// Mitsubishi GX Works2 project: LD_windingmachine   PLC: FX1N/FX1NC

PROGRAM MAIN
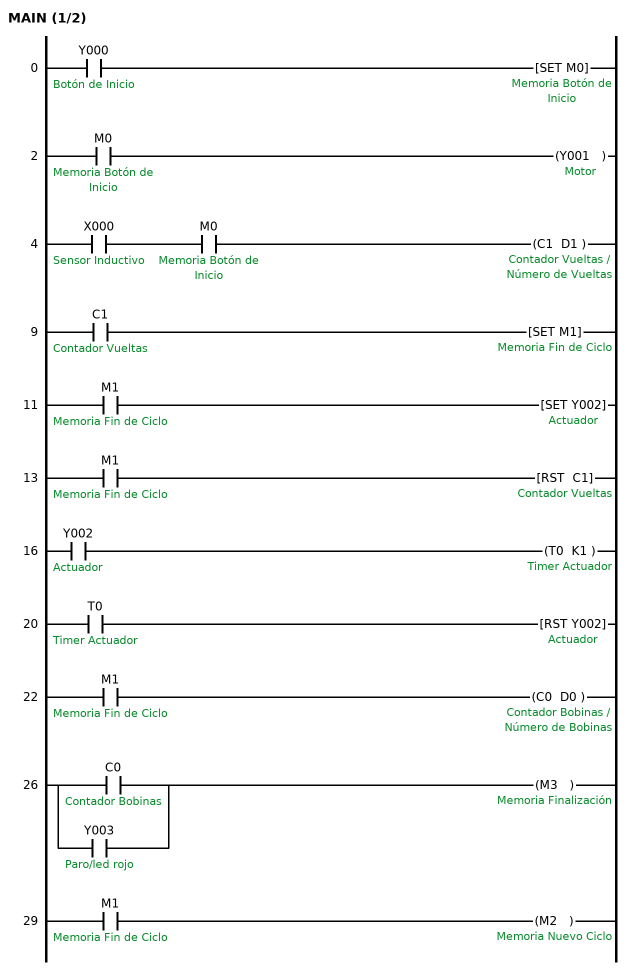
0     LD      Y000  ; Botón de Inicio
      SET     M0  ; Memoria Botón de Inicio
2     LD      M0  ; Memoria Botón de Inicio
      OUT     Y001  ; Motor
4     LD      X000  ; Sensor Inductivo
      AND     M0  ; Memoria Botón de Inicio
      OUT     C1 D1  ; Contador Vueltas / Número de Vueltas
9     LD      C1  ; Contador Vueltas
      SET     M1  ; Memoria Fin de Ciclo
11    LD      M1  ; Memoria Fin de Ciclo
      SET     Y002  ; Actuador
13    LD      M1  ; Memoria Fin de Ciclo
      RST     C1  ; Contador Vueltas
16    LD      Y002  ; Actuador
      OUT     T0 K1  ; Timer Actuador
20    LD      T0  ; Timer Actuador
      RST     Y002  ; Actuador
22    LD      M1  ; Memoria Fin de Ciclo
      OUT     C0 D0  ; Contador Bobinas / Número de Bobinas
26    LD      C0  ; Contador Bobinas
      OR      Y003  ; Paro/led rojo
      OUT     M3  ; Memoria Finalización
29    LD      M1  ; Memoria Fin de Ciclo
      OUT     M2  ; Memoria Nuevo Ciclo
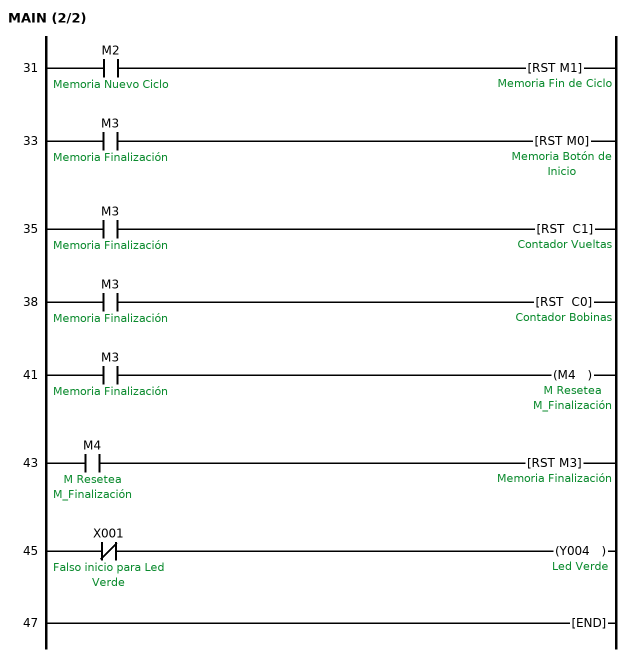
31    LD      M2  ; Memoria Nuevo Ciclo
      RST     M1  ; Memoria Fin de Ciclo
33    LD      M3  ; Memoria Finalización
      RST     M0  ; Memoria Botón de Inicio
35    LD      M3  ; Memoria Finalización
      RST     C1  ; Contador Vueltas
38    LD      M3  ; Memoria Finalización
      RST     C0  ; Contador Bobinas
41    LD      M3  ; Memoria Finalización
      OUT     M4  ; M Resetea M_Finalización
43    LD      M4  ; M Resetea M_Finalización
      RST     M3  ; Memoria Finalización
45    LDI     X001  ; Falso inicio para Led Verde
      OUT     Y004  ; Led Verde
47    END
END_PROGRAM
